DATA_BLOCK "DB"
{ S7_Optimized_Access := 'true' }
    VAR
        cnt: LINT;
        first: BOOL;
        curTimerValue: TIME;
        state0: STATE;
        curTime: LREAL;
        loopsKilled: LINT;
        curTimer: INT;
    END_VAR
BEGIN
    first := TRUE;
END_DATA_BLOCK
